// TwinCAT 3 PLC project Base
// ProgramVersion: 3.1.4022.4
// libraries:
//   Tc2_Standard, * (Beckhoff Automation GmbH)
//   Tc2_System, * (Beckhoff Automation GmbH)
//   Tc2_Utilities, * (Beckhoff Automation GmbH)
//   Tc3_IotBase, * (Beckhoff Automation GmbH)
//   Tc3_IotCommunicator, * (Beckhoff Automation GmbH)
//   Tc3_JsonXml, * (Beckhoff Automation GmbH)
//   Tc3_Module, * (Beckhoff Automation GmbH)
// project tree:
//   DUTs/ E_JsonStates.TcDUT, ST_ReceivedData.TcDUT (not stored)
//   GVLs/ CELL_STATE.TcGVL, CELL_WORKING_STATES.TcGVL (not stored), CLAMP_STATE.TcGVL (not stored), CELL_ACTION_STATE.TcGVL (not stored), DATA_SERVICE_STATE.TcGVL, MHS_STATE.TcGVL (not stored), MHS_Registers.TcGVL (not stored)
//   / PlcTask.TcTTO
//   POUs/ FB_Bool_To_Word.TcPOU, FB_Cell_Simu.TcPOU (not stored), FB_InterfaceProfibus.TcPOU, FB_VirtualCell.TcPOU, FB_Word_To_Bool.TcPOU, I_CELL.TcIO (not stored), FB_Cell.TcPOU (not stored), FB_Clamp.TcPOU (not stored), FB_ClampSimulated.TcPOU (not stored), FB_DataService.TcPOU (not stored), FB_InterfaceIO.TcPOU, FB_InterfaceSimulated.TcPOU (not stored), FB_MHS.TcPOU, ITF_Cell.TcIO, JsonSaxHandler.TcPOU, MAIN.TcPOU (not stored), FB_VirtualCellIntWriter.TcPOU
//   POUs/REST API/MHS/ FB_Get.TcPOU, FB_PUT.TcPOU
// real-time tasks:
//   TASK PlcTask: cycle T#10ms, priority 20, ADS port 350
// I/O:
//   DEVICE Device 3 (EtherCAT), AmsNetId 192.168.74.113.4.1
//     Box 1 (CU1128) [CU1128 6x EtherCAT junction]
//       A2_Schaltschrank [EK1100 EtherCAT Coupler (2A E-Bus)]
//         Term 3 (EL2004) [EL2004 4Ch. Dig. Output 24V, 0.5A]
//         Term 4 (EL1004) [EL1004 4Ch. Dig. Input 24V, 3ms]
//         Term 5 (EL2004) [EL2004 4Ch. Dig. Output 24V, 0.5A]
//         Term 6 (EL2004) [EL2004 4Ch. Dig. Output 24V, 0.5A]
//         Term 7 (EL1004) [EL1004 4Ch. Dig. Input 24V, 3ms]
//         Term 8 (EL1004) [EL1004 4Ch. Dig. Input 24V, 3ms]
//         Term 9 (EL2004) [EL2004 4Ch. Dig. Output 24V, 0.5A]
//         Term 10 (EL1004) [EL1004 4Ch. Dig. Input 24V, 3ms]
//         Term 24 (EL9011) [EL9011 End Terminal]
//       A5 [EK1100 EtherCAT Coupler (2A E-Bus)]
//         Term 12 (EL1004) [EL1004 4Ch. Dig. Input 24V, 3ms]
//         Term 13 (EL1004) [EL1004 4Ch. Dig. Input 24V, 3ms]
//         Term 14 (EL2004) [EL2004 4Ch. Dig. Output 24V, 0.5A]
//         Term 15 (EL2004) [EL2004 4Ch. Dig. Output 24V, 0.5A]
//         Term 16 (EL2004) [EL2004 4Ch. Dig. Output 24V, 0.5A]
//         Term 25 (EL9011) [EL9011 End Terminal]
//       Dummy term [CU1128 6x EtherCAT junction - Dev A]
//         Term 18 (EK1100) [EK1100 EtherCAT Coupler (2A E-Bus)]
//           Term 19 (EL1004) [EL1004 4Ch. Dig. Input 24V, 3ms]
//           Term 20 (EL9505) [EL9505 Power supply terminal 5V]
//           Term 21 (EL1124) [EL1124 4Ch. Dig. Input 5V, 10µs, Sensor Power]
//           Term 22 (EL2124) [EL2124 4Ch. Dig. Output 5V, 20mA]
//           Term 26 (EL9011) [EL9011 End Terminal]
//       Term 25 (CU1128-C) [CU1128 6x EtherCAT junction - Dev B]
// variable links:
//   Base/Base Instance <-> Device 3 (EtherCAT)/Box 1 (CU1128)/A2_Schaltschrank/Term 3 (EL2004)
//     PlcTask Outputs/MAIN.fbCellA2.fbClamp.m_bOpen <-> Channel 1/NPSA2
//   Base/Base Instance <-> Device 3 (EtherCAT)/Box 1 (CU1128)/A2_Schaltschrank/Term 4 (EL1004)
//     PlcTask Inputs/MAIN.fbCellA2.fbClamp.m_bIsClosed <-> Channel 1/A2_NPS_Gespannt
//     PlcTask Inputs/MAIN.fbCellA2.fbClamp.m_bIsFull <-> Channel 3/A2_NPS_Ini_Oben
//     PlcTask Inputs/MAIN.fbCellA2.fbClamp.m_bIsOpen <-> Channel 2/A2_NPS_Auf
//   Base/Base Instance <-> Device 3 (EtherCAT)/Box 1 (CU1128)/A2_Schaltschrank/Term 5 (EL2004)
//     PlcTask Outputs/MAIN.fbCellA2.fbInterface.m_bMoveToLoadPos <-> Channel 1/A2_Bestück
//     PlcTask Outputs/MAIN.fbCellA2.fbInterface.m_bMoveToUnloadPos <-> Channel 3/A2_Entnahme
//     PlcTask Outputs/MAIN.fbCellA2.fbInterface.m_bStart <-> Channel 2/A2_Startfreigabe
//     PlcTask Outputs/MAIN.fbCellA2.fbInterface.m_bToStandby <-> Channel 4/A2_Standby
//   Base/Base Instance <-> Device 3 (EtherCAT)/Box 1 (CU1128)/A2_Schaltschrank/Term 7 (EL1004)
//     PlcTask Inputs/MAIN.fbCellA2.fbInterface.m_bFinished <-> Channel 3/A2_Fertig
//     PlcTask Inputs/MAIN.fbCellA2.fbInterface.m_bLoadPos <-> Channel 1/A2_Bestückbereit
//     PlcTask Inputs/MAIN.fbCellA2.fbInterface.m_bRunning <-> Channel 2/A2_Arbeitet
//     PlcTask Inputs/MAIN.fbCellA2.fbInterface.m_bUnloadPos <-> Channel 4/A2_Entnahmebereit
//   Base/Base Instance <-> Device 3 (EtherCAT)/Box 1 (CU1128)/A2_Schaltschrank/Term 8 (EL1004)
//     PlcTask Inputs/MAIN.fbCellA2.fbInterface.m_bEmergencyOff <-> Channel 4/Input
//     PlcTask Inputs/MAIN.fbCellA2.fbInterface.m_bStandby <-> Channel 1/Input
//   Base/Base Instance <-> Device 3 (EtherCAT)/Box 1 (CU1128)/A5/Term 12 (EL1004)
//     PlcTask Inputs/MAIN.fbCellA5.fbInterface.m_bFinished <-> Channel 3/A5_Fertig
//     PlcTask Inputs/MAIN.fbCellA5.fbInterface.m_bLoadPos <-> Channel 1/A5_Bestückbereit
//     PlcTask Inputs/MAIN.fbCellA5.fbInterface.m_bRunning <-> Channel 2/A5_Arbeitet
//     PlcTask Inputs/MAIN.fbCellA5.fbInterface.m_bUnloadPos <-> Channel 4/A5_Entnahmebereit
//   Base/Base Instance <-> Device 3 (EtherCAT)/Box 1 (CU1128)/A5/Term 13 (EL1004)
//     PlcTask Inputs/MAIN.fbCellA5.fbClamp.m_bIsClosed <-> Channel 3/A5_NPS_Zu
//     PlcTask Inputs/MAIN.fbCellA5.fbClamp.m_bIsFull <-> Channel 1/A5_NPS_Ini_Oben
//     PlcTask Inputs/MAIN.fbCellA5.fbClamp.m_bIsOpen <-> Channel 2/A5_NPS_Auf
//   Base/Base Instance <-> Device 3 (EtherCAT)/Box 1 (CU1128)/A5/Term 14 (EL2004)
//     PlcTask Outputs/MAIN.fbCellA5.fbInterface.m_bMoveToLoadPos <-> Channel 1/A5_Bestückposition
//     PlcTask Outputs/MAIN.fbCellA5.fbInterface.m_bMoveToUnloadPos <-> Channel 3/A5_Fahre_Entnahmeposition
//     PlcTask Outputs/MAIN.fbCellA5.fbInterface.m_bStart <-> Channel 2/A5_Startfreigabe
//     PlcTask Outputs/MAIN.fbCellA5.fbInterface.m_bToStandby <-> Channel 4/A5_Fahre_Standby
//   Base/Base Instance <-> Device 3 (EtherCAT)/Box 1 (CU1128)/A5/Term 15 (EL2004)
//     PlcTask Outputs/MAIN.fbCellA5.fbClamp.m_bOpen <-> Channel 1/A5_NPS

CONFIGURATION Base
    RESOURCE PLC ON TwinCAT3
        TASK PlcTask(INTERVAL := T#10ms, PRIORITY := 20);
        PROGRAM MAIN WITH PlcTask : MAIN;
    END_RESOURCE
END_CONFIGURATION

// ---- DUTs/E_JsonStates.TcDUT
{attribute 'qualified_only'}
{attribute 'strict'}
TYPE E_JsonStates :
(
	JSON_STATE_ONSTARTOBJECT1 := 10,
	JSON_STATE_ONKEY_VALUES := 20,
	
	JSON_STATE_ONKEY_ACTIONID := 11,
	JSON_STATE_ONSTRING1 := 12,
	JSON_STATE_ONKEY_WPID := 30,
	JSON_STATE_ONSTRING2 := 40,
	JSON_STATE_ONKEY_WPPLACE := 50,
	JSON_STATE_ONDINT1 := 60,
	JSON_STATE_ONKEY_CELL := 70,
	JSON_STATE_ONUDINT2 := 80,
	JSON_STATE_ONKEY_ACTIONTYPE := 90,
	JSON_STATE_ONUDINT3 := 100,
	JSON_STATE_ONKEY_ACTIONSTATE := 110,
	JSON_STATE_ONUDINT4 := 120,
	JSON_STATE_ONENDOBJECT2 := 1100,
	JSON_STATE_FINISH := 1200
);
END_TYPE

// ---- GVLs/CELL_STATE.TcGVL
{attribute 'qualified_only'}
VAR_GLOBAL
	

			
TYPE 
	CELL_STATE: (e_IDEL, e_WORKING, e_MHS_ACTION, e_ERROR );			
END_TYPE



END_VAR

// ---- GVLs/DATA_SERVICE_STATE.TcGVL
{attribute 'qualified_only'}
VAR_GLOBAL
TYPE
	DATA_SERVICE_STATE: (e_IDLE, e_BUSY, e_FINISHED, e_ERROR);	
END_TYPE
	
END_VAR

// ---- POUs/ITF_Cell.TcIO
INTERFACE ITF_Cell

METHOD GetEmergencyOff : BOOL
VAR_INPUT
END_VAR
END_METHOD

METHOD GetEmergencyStop : BOOL
VAR_INPUT
END_VAR
END_METHOD

METHOD GetFinished : BOOL
VAR_INPUT
END_VAR
END_METHOD

METHOD GetIsRunning : BOOL
VAR_INPUT
END_VAR
END_METHOD

METHOD GetLoadPos : BOOL
VAR_INPUT
END_VAR
END_METHOD

METHOD GetStandby : BOOL
VAR_INPUT
END_VAR
END_METHOD

METHOD GetStartable : BOOL
VAR_INPUT
END_VAR
END_METHOD

METHOD GetUnloadPos : BOOL
VAR_INPUT
END_VAR
END_METHOD

METHOD SetEmergencyOff : BOOL
VAR_INPUT
	b :BOOL;
END_VAR
END_METHOD

METHOD SetEmergencyStop : BOOL
VAR_INPUT
	b :BOOL;
END_VAR
END_METHOD

METHOD SetMoveToLoad : BOOL
VAR_INPUT
	b :BOOL;
END_VAR
END_METHOD

METHOD SetMoveToUnload : BOOL
VAR_INPUT
	b :BOOL;
END_VAR
END_METHOD

METHOD SetStandby : BOOL
VAR_INPUT
	b :BOOL;
END_VAR
END_METHOD

METHOD SetStart : BOOL
VAR_INPUT
	b :BOOL;
END_VAR
END_METHOD

END_INTERFACE

// ---- POUs/FB_Bool_To_Word.TcPOU
FUNCTION_BLOCK FB_Bool_To_Word
VAR_INPUT
//*Hami* Eingang Von FB	als Array Of Bool
	i_Bool : ARRAY [0..15] OF BOOL ;
END_VAR
VAR_OUTPUT
//*Hami* Ausgang Von FB	als UINT
	o_Word : UINT;
END_VAR
VAR
END_VAR

//////////////////////////////////////////////////////////////////////////////////////////////
//*Hami* Diese Funktionsbaustein kann ein Array Of Bool bekommen und in UINT dekodieren
//*Hami* Aufruf von jeder Index von UINT mit UINT.X in Compiler  möglich ist
o_Word.0 := i_Bool[0];
o_Word.1 := i_Bool[1];
o_Word.2 := i_Bool[2];
o_Word.3 := i_Bool[3];
o_Word.4 := i_Bool[4];
o_Word.5 := i_Bool[5];
o_Word.6 := i_Bool[6];
o_Word.7 := i_Bool[7];
o_Word.8 := i_Bool[8];
o_Word.9 := i_Bool[9];
o_Word.10 := i_Bool[10];
o_Word.11 := i_Bool[11];
o_Word.12 := i_Bool[12];
o_Word.13 := i_Bool[13];
o_Word.14 := i_Bool[14];
o_Word.15 := i_Bool[15];
//////////////////////////////////////////////////////////////////////////////////////////////

END_FUNCTION_BLOCK

// ---- POUs/FB_InterfaceProfibus.TcPOU
FUNCTION_BLOCK FB_InterfaceProfibus IMPLEMENTS ITF_Cell
VAR_INPUT

END_VAR
VAR_OUTPUT
END_VAR

VAR
	// Ausgang :engine          AT %IX0.0:        BOOL; 
//Eingänge
//A5Q_Bestuckung AT %QX27.4 : BOOL;
//A5Q_Startfreigabe AT %QX27.5 : BOOL;
//A5Q_Entnahme AT %QX27.6 : BOOL;
//A5Q_Standby AT %QX27.7 : BOOL;
//A5Q_NOT_Aus_Befehl AT %QX28.0 : BOOL;

//INPUTS  A5 Station Variabel : 5V Von Arduino

//A5I_Bestuckbereit_o1 AT %IX43.2 : BOOL;  
//A5I_Arbeitet_o2 AT %IX43.3 : BOOL;
//A5I_Fertig_o3 AT %IX43.4 : BOOL;
//A5I_Storung_o5 AT %IX43.5 : BOOL;
//A5I_NOT_Halt_o6 AT %IX43.6 : BOOL;
//A5I_Pro_Standby_o7 AT %IX43.7 : BOOL;
//A5I_Pro_Standby_o8 AT %IX44.0 : BOOL;
/////////////////////////////////////////////////////////////////////////////////////////////////////////////////
//*Hami* boolesche Eingänge und Ausgänge als innere Variable deklarieren 

//*Hami* innere Eingänge
m_bEmergencyOff  : BOOL; 
m_bEmergencyStop : BOOL;
m_bFinished : BOOL;
m_bRunning : BOOL;
m_bLoadPos  : BOOL; 
m_bUnloadPos  : BOOL; 
m_bStandby : BOOL;
m_bStartable : BOOL;
m_bSoftError  : BOOL;

//*Hami* innere Ausgänge
m_bToEmergencyOff  : BOOL;
m_bToEmergencyStop  : BOOL;
m_bMoveToLoadPos  : BOOL;
m_bMoveToUnloadPos : BOOL;
m_bToStandby  : BOOL;
m_bStart  : BOOL;

//*HAMI* Eingäng und Ausgäng in Form UINT deklarieren zum anpassen Profibus_Dateien
//*HAMI* Die beide müssen zu ProfibusKlemme gelinkt werden

m_wProfibusDataWord AT %I*  : UINT; 
m_wToProfibusDataWord AT %Q*  : UINT;

//*HAMI* Hilf_FBs Deklarieren (Konvertor)

fbBoolToWord : FB_Bool_To_Word;
fbWordToBool : FB_Word_To_Bool;
//*HAMI* Variable für Konvertor FBs ( FB_Bool_to_Word und FB_Word_to_bool )
//*HAMI* i_arrayOfBool Eingänge q_arrayOfBool Ausgänge
i_arrayOfBool : ARRAY [0..15] OF BOOL;
q_arrayOfBool : ARRAY [0..15] OF BOOL;
//*Hami physikalische Eingänge und Ausgänge von Profibus werden drin geschrieben *
i_DataWord : UINT ;
q_DataWord : UINT ;
/////////////////////////////////////////////////////////////////////////////////////////////////////////////////


END_VAR

/////////////////////////////////////////////////////////////////////////////////////////////////////////////////
//*Hami* Aufruf von Hilf_FBs (Konvertor) 
fbBoolToWord();
fbWordToBool();


//hier Wird Mit Hilfe Von Funktion Blocks ( FB_Bool_to_Word und FB_Word_to_bool ) eingänge und Ausgänge angepasst

// Eingänge von Zelle To Bool
i_DataWord := m_wProfibusDataWord ;  //*Hami* Eingang von Profibus in einem hilfsvariabel schreiben
fbWordToBool.i_Word := i_DataWord ; //*Hami* Eingang von Profibus in Eingang von FB_WordToBool schreiben 
i_arrayOfBool :=fbWordToBool.o_Bool ; //*Hami* Ausgang von FB_WordToBool in ein Array of Bool Schreiben 


//*Hami* jeder Index von Array wurde gleich innere Eingänge gestellt 
m_bEmergencyOff := i_arrayOfBool[0];
m_bEmergencyStop := i_arrayOfBool[1]; 
m_bFinished := i_arrayOfBool[2];
m_bRunning := i_arrayOfBool[3];
m_bLoadPos := i_arrayOfBool[4]; 
m_bUnloadPos := i_arrayOfBool[5];   
m_bStandby := i_arrayOfBool[6];
m_bStartable := i_arrayOfBool[7];
m_bSoftError := i_arrayOfBool[8];

//*Hami* Ausgänge von Zelle To Array of Bool 

q_arrayOfBool[0]:= m_bToEmergencyOff ;
q_arrayOfBool[1] := m_bToEmergencyStop;  
q_arrayOfBool[2] := m_bMoveToLoadPos;  
q_arrayOfBool[3] := m_bMoveToUnloadPos; 
q_arrayOfBool[4] := m_bToStandby;  
q_arrayOfBool[5] := m_bStart;

fbBoolToWord.i_Bool := q_arrayOfBool ;//*Hami* Array of Bool in Eingang von fbBoolToWord schreiben
q_DataWord := fbBoolToWord.o_Word ;  //*Hami*  Ausgang von FB_BoolToWord in einem Hilfsvariabel schreiben 
m_wToProfibusDataWord := q_DataWord ; //*Hami* Hilfsvariabel in Ausgang von Profibus Schreiben

/////////////////////////////////////////////////////////////////////////////////////////////////////////////////


// Logik des Interfaces in diesem Fall zurücksetzen der Ausgänge nach erreichen des Ziels 
// Aus Zustandsmaschine Löschen ggf. ??
//IF m_bEmergencyOff THEN
//m_bToEmergencyOff := FALSE;
//END_IF

//IF m_bEmergencyStop THEN
//m_bToEmergencyStop := FALSE;
//END_IF

IF m_bLoadPos THEN
	m_bMoveToLoadPos := FALSE;
END_IF

IF m_bUnloadPos THEN
	m_bMoveToUnloadPos := FALSE;
END_IF

IF m_bStandby THEN
	m_bToStandby := FALSE;
END_IF

IF m_bRunning THEN
	m_bStart := FALSE;
END_IF

METHOD GetEmergencyOff : BOOL
VAR_INPUT
END_VAR
GetEmergencyOff := m_bEmergencyOff;
END_METHOD

METHOD GetEmergencyStop : BOOL
VAR_INPUT
END_VAR
GetEmergencyStop := m_bEmergencyStop;
END_METHOD

METHOD GetFinished : BOOL
VAR_INPUT
END_VAR
GetFinished := m_bFinished;
END_METHOD

METHOD GetIsRunning : BOOL
VAR_INPUT
END_VAR
GetIsRunning := m_bRunning;
END_METHOD

METHOD GetLoadPos : BOOL
VAR_INPUT
END_VAR
GetLoadPos := m_bLoadPos;
END_METHOD

METHOD GetStandby : BOOL
VAR_INPUT
END_VAR
GetStandby := m_bStandby;
END_METHOD

METHOD GetStartable : BOOL
VAR_INPUT
END_VAR
GetStartable := m_bStartable;
END_METHOD

METHOD GetUnloadPos : BOOL
VAR_INPUT
END_VAR
GetUnloadPos := m_bUnloadPos;
END_METHOD

METHOD SetEmergencyOff : BOOL
VAR_INPUT
	b :BOOL;
END_VAR

m_bToEmergencyOff := b;
SetEmergencyOff:=b;
END_METHOD

METHOD SetEmergencyStop : BOOL
VAR_INPUT
	b :BOOL;
END_VAR
m_bToEmergencyStop :=b;

SetEmergencyStop := b;
END_METHOD

METHOD SetMoveToLoad : BOOL
VAR_INPUT
	b :BOOL;
END_VAR
m_bMoveToLoadPos := b;

SetMoveToLoad := b;
END_METHOD

METHOD SetMoveToUnload : BOOL
VAR_INPUT
	b :BOOL;
END_VAR
m_bMoveToUnloadPos := b;

SetMoveToUnload := b;
END_METHOD

METHOD SetStandby : BOOL
VAR_INPUT
	b :BOOL;
END_VAR
m_bToStandby := b;

SetStandby := b;
END_METHOD

METHOD SetStart : BOOL
VAR_INPUT
	b :BOOL;
END_VAR
m_bStart := b;

SetStart := b;
END_METHOD

END_FUNCTION_BLOCK

// ---- POUs/FB_Word_To_Bool.TcPOU
FUNCTION_BLOCK FB_Word_To_Bool
VAR_INPUT
//*Hami* Eingang Von FB	als UINT
	i_Word : UINT;
END_VAR
VAR_OUTPUT
//*Hami* Ausgang Von FB	als Array
	o_Bool : ARRAY [0..15] OF BOOL ;
END_VAR
VAR
END_VAR

//////////////////////////////////////////////////////////////////////////////////////////////
//*Hami* Diese Funktionsbaustein kann ein UINT bekommen und in Array Of Bool dekodieren
//*Hami* Aufruf von jeder Index von UINT mit UINT.X in Compiler  möglich ist
o_Bool[0] := i_Word.0 ;
o_Bool[1] := i_Word.1 ;
o_Bool[2] := i_Word.2 ;
o_Bool[3] := i_Word.3 ;
o_Bool[4] := i_Word.4 ;
o_Bool[5] := i_Word.5 ;	
o_Bool[6] := i_Word.6 ;
o_Bool[7] := i_Word.7 ;
o_Bool[8] := i_Word.8 ;
o_Bool[9] := i_Word.9 ;
o_Bool[10] := i_Word.10 ;
o_Bool[11] := i_Word.11 ;
o_Bool[12] := i_Word.12 ;
o_Bool[13] := i_Word.13 ;
o_Bool[14] := i_Word.14 ;
o_Bool[15] := i_Word.15 ;
//////////////////////////////////////////////////////////////////////////////////////////////

END_FUNCTION_BLOCK

// ---- POUs/FB_VirtualCell.TcPOU
FUNCTION_BLOCK FB_VirtualCell IMPLEMENTS I_CELL
VAR_INPUT
	
END_VAR
VAR_OUTPUT
END_VAR
VAR
	m_csStateRequest : CELL_ACTION_STATE;
	m_csStateRequestOld : CELL_ACTION_STATE;
	m_csState : CELL_ACTION_STATE;
	m_csStateLastCycle : CELL_ACTION_STATE;
	m_csStateLastAction : CELL_ACTION_STATE;
	
	
	m_csSRWorkingState : CELL_WORKING_STATES := CELL_WORKING_STATES.e_FINISHED;
	m_csSRWorkingStateLast : CELL_WORKING_STATES := CELL_WORKING_STATES.e_FINISHED;
	// Eigenschaften
	m_sName : STRING;
	m_bIsDisassemblyCell : BOOL;
	
	m_iWorkpiece : DINT;
	m_sWorkpieceID : STRING;
	

	m_csCellState : CELL_STATE;
	m_csCellStateLast : CELL_STATE;


	
	m_sErrorString : STRING;
	
	// DataServices
	

	m_sConfigString : STRING;
	m_sConfigStringEndGet : STRING  := '_Get.exe';
	m_sConfigStringEndPut : STRING  := '_Put.exe';
	
	// Virtuelle Zellen Verbindung
	fbVirtualCellIntWriter 	: FB_VirtualCellIntWriter;
	fbJson      			: FB_JsonSaxWriter;
	m_sJsonAction 			: STRING;
	m_sActionPath 			: STRING;
	m_sActionName			: STRING;
	m_sActionPathDir 		: STRING   := 'C:\Sysdem\Netzwerklaufwerk_19-0011';
	m_sAMSNetID 			: 	STRING 	:=	'192.168.74.113.1.1';
	
END_VAR

METHOD GetErrorString : STRING
VAR_INPUT
END_VAR
END_METHOD

METHOD GetName : STRING
VAR_INPUT
END_VAR
GetName := m_sName;
END_METHOD

METHOD PUBLIC GetState : INT
VAR_INPUT
	
END_VAR
GetState := CELL_ACTION_STATE.e_Standby;
END_METHOD

METHOD GetWorkpiece : DINT
VAR_INPUT
END_VAR
GetWorkpiece := m_iWorkpiece;
END_METHOD

METHOD IsDisassemblyCell : BOOL
VAR_INPUT
END_VAR
IsDisassemblyCell := FALSE; // Kann keine sein ist virtuell
END_METHOD

METHOD IsError : BOOL
VAR_INPUT
END_VAR
IF m_csCellState = CELL_STATE.e_ERROR THEN
	IsError := TRUE;
END_IF
END_METHOD

METHOD IsIdle : BOOL
VAR_INPUT
END_VAR
IF m_csCellState = CELL_STATE.e_IDEL THEN
	IsIdle := TRUE;
END_IF
END_METHOD

METHOD IsVirtualCell : BOOL
VAR_INPUT
END_VAR
IsVirtualCell :=TRUE;
END_METHOD

METHOD PUBLIC RequestActionState : BOOL
VAR_INPUT
	csStateRequest : CELL_ACTION_STATE;
END_VAR
m_csStateRequest := csStateRequest;
END_METHOD

METHOD RequestWork : BOOL
VAR_INPUT
END_VAR
m_csCellState := CELL_STATE.e_WORKING;
END_METHOD

METHOD SetDisassemblyCell : BOOL
VAR_INPUT
	bIsDisassemblyCell : BOOL;
END_VAR
m_bIsDisassemblyCell := bIsDisassemblyCell;
END_METHOD

METHOD SetGetDataServiceEnable : BOOL
VAR_INPUT
END_VAR

SetGetDataServiceEnable := FALSE;
END_METHOD

METHOD SetName : BOOL
VAR_INPUT
	sName :string ;
END_VAR
m_sName := sName;
END_METHOD

METHOD SetPutDataServiceEnable : BOOL
VAR_INPUT
END_VAR

SetPutDataServiceEnable := FALSE;
END_METHOD

METHOD SetVirtualCell : BOOL
VAR_INPUT
END_VAR
END_METHOD

METHOD SetWorkpiece : BOOL
VAR_INPUT
	iWorkpiece : DINT;
	sWorkpieceID : STRING;
END_VAR
m_iWorkpiece := iWorkpiece;
m_sWorkpieceID := sWorkpieceID;
END_METHOD

METHOD PUBLIC StateMachine : BOOL
VAR_INPUT
END_VAR

//Zellen Zustandsmaschine

CASE m_csCellState OF 
	CELL_STATE.e_IDEL:
			
	
		;
 	CELL_STATE.e_MHS_ACTION;
		//SubRoutine für Aktion beim beladen aktuell leer da keine MHS für eine virtuelle Zelle verfügbar sind 
		;
	CELL_STATE.e_WORKING:
		//SubRoutine zum Durchführen einer Bearbeitung
			//Erstellen des Json-Strings für die Datei		
			fbJson.ResetDocument();
		
			fbJson.StartObject();
            fbJson.AddKey('Name');
			fbJson.AddString(m_sName);
			fbJson.AddKey('WPID');
			fbJson.AddString(m_sWorkpieceID);			
			fbJson.EndObject();
			m_sJsonAction := fbJson.GetDocument();
		
			// Phad der Schnittstellen-Datei
			m_sActionPath := CONCAT (m_sActionPathDir,'\');
			m_sActionPath := CONCAT (m_sActionPath, m_sName);
			m_sActionPath := CONCAT (m_sActionPath, '_');
			m_sActionPath := CONCAT (m_sActionPath, m_sWorkpieceID);
			m_sActionPath := CONCAT (m_sActionPath, '.json');
			
			// Name der Schnittstellen-Datei
			m_sActionName := CONCAT (m_sName, '_');
			m_sActionName := CONCAT (m_sActionName, m_sWorkpieceID);
			m_sActionName := CONCAT (m_sActionName, '.json');
			
			// Nächster Schritt SubRoutine Starten um das Schreiben auszugühren
			IF NOT (CELL_STATE.e_WORKING = m_csCellStateLast) THEN  
				m_csSRWorkingState := CELL_WORKING_STATES.e_START;
			END_IF

			
	CASE m_csSRWorkingState OF
			
			CELL_WORKING_STATES.e_START:
				fbVirtualCellIntWriter.buffRead := m_sJsonAction; // Inhalt der Datei übergeben
				fbVirtualCellIntWriter.sDestPathName := m_sActionPath; // Pfad der Datei
				fbVirtualCellIntWriter.sDestNetId := m_sAMSNetID;// Net Id des HostPC
				fbVirtualCellIntWriter.tTimeOut := DEFAULT_ADS_TIMEOUT;// Fehlerzeit
				fbVirtualCellIntWriter.bExecute := TRUE;// Positive flanke zum Starten
				IF fbVirtualCellIntWriter.bError THEN//
					m_csCellState := CELL_STATE.e_ERROR;
				END_IF
				IF fbVirtualCellIntWriter.bBusy THEN // Der Funktionsblock aufgehört hat zu arbeiten nächster Schritt ggf. das vorhanden sein der Datei prüfen 
					
					m_csSRWorkingState := CELL_WORKING_STATES.e_WORKING;
				END_IF
				

				
			CELL_WORKING_STATES.e_WORKING:	
				fbVirtualCellIntWriter.bExecute := FALSE; // Nur positive Flanke
				IF NOT(fbVirtualCellIntWriter.bBusy) THEN // Der Funktionsblock aufgehört hat zu arbeiten nächster Schritt ggf. das vorhanden sein der Datei prüfen 
					
					m_csSRWorkingState := CELL_WORKING_STATES.e_FINISHED;
				END_IF
				
			CELL_WORKING_STATES.e_FINISHED:
				m_iWorkpiece := 0;
				m_sWorkpieceID := 'Empty';
				m_csCellState := CELL_STATE.e_IDEL;
			
		END_CASE
		
	CELL_STATE.e_ERROR:
			;
END_CASE

m_csCellStateLast := m_csCellState;
fbVirtualCellIntWriter();
fbVirtualCellIntWriter.StateMachine();
END_METHOD

METHOD StateMachineProfibus : BOOL
VAR_INPUT
END_VAR
END_METHOD

END_FUNCTION_BLOCK

// ---- POUs/FB_VirtualCellIntWriter.TcPOU
FUNCTION_BLOCK FB_VirtualCellIntWriter
VAR_INPUT
     
        sDestNetId              : T_AmsNetId;(* TwinCAT network address of the destination file *)
        sDestPathName           : T_MaxString; (* Destination file path and name *)
        bExecute                : BOOL; (* Rising edge start fb execution *)
        tTimeOut                : TIME := DEFAULT_ADS_TIMEOUT;(* Max. ADS timeout time *)
		buffRead                : STRING;// ARRAY[1..1000] OF BYTE;(* Buffer *)
END_VAR
VAR_OUTPUT
        bBusy                   :BOOL;(* TRUE => File copy execution in progress, FALSE => File copy execution idle *)
 		bError                  :BOOL;(* TRUE => Error, FALSE => No error *)
 		nErrId                  :UDINT;(* Error code *)
END_VAR
VAR
        fbFileOpen              :FB_FileOpen;
        fbFileClose             :FB_FileClose;
        fbFileRead              :FB_FileRead;
        fbFileWrite             :FB_FileWrite;

        hSrcFile                :UINT   := 0;(* File handle of the source file *)
 		hDestFile               :UINT   := 0;(* File handle of the destination file *)

        Step                    :DWORD;
        RisingEdge              :R_TRIG;

        
 		cbReadLength            :UDINT := 0;
END_VAR

METHOD StateMachine : BOOL
VAR_INPUT
END_VAR
RisingEdge(CLK:=bExecute);

CASE Step OF
        0:      (* Idle state *)
         IF RisingEdge.Q THEN
                        bBusy := TRUE;
                        bError:= FALSE;
                        nErrId:=0;
                        Step := 1;
                        cbReadLength:=0;
                        hSrcFile:=0;
                        hDestFile:=0;
                END_IF



        1:      (* Open destination file *)
         fbFileOpen( bExecute := FALSE );
                fbFileOpen( sNetId := sDestNetId, sPathName := sDestPathName,
                        nMode := FOPEN_MODEWRITE OR FOPEN_MODEBINARY,
                        ePath := PATH_GENERIC, tTimeout := tTimeOut, bExecute := TRUE );
                Step := Step+1;
        2:
                fbFileOpen( bExecute := FALSE );
                IF NOT fbFileOpen.bBusy THEN
                        IF fbFileOpen.bError THEN
                                nErrId := fbFileOpen.nErrId;
                                bError := TRUE;
                                Step := 50;
                        ELSE
                                hDestFile := fbFileOpen.hFile;
                                Step := Step + 1;
                        END_IF
                END_IF

        3:      (* Write data to destination file *)
         fbFileWrite( bExecute := FALSE );
                fbFileWrite( sNetId:=sDestNetId, hFile:=hDestFile,
                        pWriteBuff:= ADR(buffRead), cbWriteLen:= INT_TO_UDINT(LEN(buffRead)),
                        bExecute:=TRUE, tTimeout:=tTimeOut );
                Step := Step + 1;
				
        4:
                fbFileWrite( bExecute := FALSE );
                IF NOT fbFileWrite.bBusy THEN
                        IF fbFileWrite.bError THEN
                                nErrId := fbFileWrite.nErrId;
                                bError := TRUE;
                                Step := 50;
                        ELSE
                                 Step := 50;(* Cleanup: close the destination and source files *)
                         
                        
                        END_IF
                END_IF

        30:     (* Close the destination file *)
         fbFileClose( bExecute := FALSE );
                fbFileClose( sNetId:=sDestNetId, hFile:=hDestFile, bExecute:=TRUE, tTimeout:=tTimeOut );
                Step := Step + 1;
        31:
                fbFileClose( bExecute := FALSE );
                IF NOT fbFileClose.bBusy THEN
                        IF fbFileClose.bError THEN
                                nErrId := fbFileClose.nErrId;
                                bError := TRUE;
                        END_IF
                        Step := 50;
                        hDestFile := 0;
                END_IF

        40: (* Close source file *)
         fbFileClose( bExecute := FALSE );
               // fbFileClose( sNetId:=sSrcNetId, hFile:=hSrcFile, bExecute:=TRUE, tTimeout:=tTimeOut );
                Step := Step + 1;
        41:
                fbFileClose( bExecute := FALSE );
                IF NOT fbFileClose.bBusy THEN
                        IF fbFileClose.bError THEN
                                nErrId := fbFileClose.nErrId;
                                bError := TRUE;
                        END_IF
                        Step := 50;
                        hSrcFile := 0;
                END_IF

        50: (* Error or ready => Cleanup *)
         IF ( hDestFile <> 0 ) THEN
                        Step := 30; (* Close the destination file*)
         ELSIF (hSrcFile <> 0 ) THEN
                        Step := 40; (* Close the source file *)
         ELSE
                        Step := 0;      (* Ready *)
                        bBusy := FALSE;
                END_IF

END_CASE
END_METHOD

END_FUNCTION_BLOCK

// ---- POUs/FB_InterfaceIO.TcPOU
FUNCTION_BLOCK FB_InterfaceIO IMPLEMENTS ITF_Cell
VAR_INPUT

END_VAR
VAR_OUTPUT
END_VAR


	// Ausgang :engine          AT %IX0.0:        BOOL; 
//Eingänge
//A5Q_Bestuckung AT %QX27.4 : BOOL;
//A5Q_Startfreigabe AT %QX27.5 : BOOL;
//A5Q_Entnahme AT %QX27.6 : BOOL;
//A5Q_Standby AT %QX27.7 : BOOL;
//A5Q_NOT_Aus_Befehl AT %QX28.0 : BOOL;

//INPUTS  A5 Station Variabel : 5V Von Arduino

//A5I_Bestuckbereit_o1 AT %IX43.2 : BOOL;  
//A5I_Arbeitet_o2 AT %IX43.3 : BOOL;
//A5I_Fertig_o3 AT %IX43.4 : BOOL;
//A5I_Storung_o5 AT %IX43.5 : BOOL;
//A5I_NOT_Halt_o6 AT %IX43.6 : BOOL;
//A5I_Pro_Standby_o7 AT %IX43.7 : BOOL;
//A5I_Pro_Standby_o8 AT %IX44.0 : BOOL;
VAR
m_bEmergencyOff AT %I* : BOOL;
m_bEmergencyStop AT %I* : BOOL;
m_bFinished AT %I* : BOOL;
m_bRunning AT %I* : BOOL;
m_bLoadPos  AT %I* : BOOL; 
m_bUnloadPos  AT %I* : BOOL; 
m_bStandby AT %I* : BOOL;
m_bStartable AT %I* : BOOL;
m_bSoftError AT %I* : BOOL;
// Ausgang :engine          AT %QX0.0:        BOOL; 
// Ausgänge
m_bToEmergencyOff AT %Q* : BOOL;
m_bToEmergencyStop AT %Q* : BOOL;
m_bMoveToLoadPos AT %Q* : BOOL;
m_bMoveToUnloadPos AT %Q* : BOOL;
m_bToStandby AT %Q* : BOOL;
m_bStart AT %Q* : BOOL;

END_VAR

// Logik des Interfaces in diesem Fall zurücksetzen der Ausgänge nach erreichen des Ziels 
// Aus Zustandsmaschine Löschen ggf. ??
//IF m_bEmergencyOff THEN
//m_bToEmergencyOff := FALSE;
//END_IF

//IF m_bEmergencyStop THEN
//m_bToEmergencyStop := FALSE;
//END_IF

IF m_bLoadPos THEN
	m_bMoveToLoadPos := FALSE;
END_IF

IF m_bUnloadPos THEN
	m_bMoveToUnloadPos := FALSE;
END_IF

IF m_bStandby THEN
	m_bToStandby := FALSE;
END_IF

IF m_bRunning THEN
	m_bStart := FALSE;
END_IF

METHOD GetEmergencyOff : BOOL
VAR_INPUT
END_VAR
GetEmergencyOff := m_bEmergencyOff;
END_METHOD

METHOD GetEmergencyStop : BOOL
VAR_INPUT
END_VAR
GetEmergencyStop := m_bEmergencyStop;
END_METHOD

METHOD GetFinished : BOOL
VAR_INPUT
END_VAR
GetFinished := m_bFinished;
END_METHOD

METHOD GetIsRunning : BOOL
VAR_INPUT
END_VAR
GetIsRunning := m_bRunning;
END_METHOD

METHOD GetLoadPos : BOOL
VAR_INPUT
END_VAR
GetLoadPos := m_bLoadPos;
END_METHOD

METHOD GetStandby : BOOL
VAR_INPUT
END_VAR
GetStandby := m_bStandby;
END_METHOD

METHOD GetStartable : BOOL
VAR_INPUT
END_VAR
GetStartable := m_bStartable;
END_METHOD

METHOD GetUnloadPos : BOOL
VAR_INPUT
END_VAR
GetUnloadPos := m_bUnloadPos;
END_METHOD

METHOD SetEmergencyOff : BOOL
VAR_INPUT
	b :BOOL;
END_VAR

m_bToEmergencyOff := b;
SetEmergencyOff:=b;
END_METHOD

METHOD SetEmergencyStop : BOOL
VAR_INPUT
	b :BOOL;
END_VAR
m_bToEmergencyStop :=b;

SetEmergencyStop := b;
END_METHOD

METHOD SetMoveToLoad : BOOL
VAR_INPUT
	b :BOOL;
END_VAR
m_bMoveToLoadPos := b;

SetMoveToLoad := b;
END_METHOD

METHOD SetMoveToUnload : BOOL
VAR_INPUT
	b :BOOL;
END_VAR
m_bMoveToUnloadPos := b;

SetMoveToUnload := b;
END_METHOD

METHOD SetStandby : BOOL
VAR_INPUT
	b :BOOL;
END_VAR
m_bToStandby := b;

SetStandby := b;
END_METHOD

METHOD SetStart : BOOL
VAR_INPUT
	b :BOOL;
END_VAR
m_bStart := b;

SetStart := b;
END_METHOD

END_FUNCTION_BLOCK

// ---- POUs/FB_MHS.TcPOU
FUNCTION_BLOCK FB_MHS


VAR
	m_csStateRequest : MHS_STATE;
	m_csStateRequestOld : MHS_STATE;
	m_csState : MHS_STATE;
	m_csStateLastCycle : MHS_STATE;
	m_csStateLastAction : MHS_STATE;
	m_Name : STRING;	
	// Von SystemDemonstratorApp kommend
	m_iWorkpiece : DINT; 
	m_iCell : DINT;
	m_iRequest: DINT;
	// Von SystemDemonstratorApp kommend angenommen
	m_iWorkpieceAccepted : DINT; 
	m_iCellAccepted : DINT;
	m_iRequestAccepted: DINT;
	
	// Von PLC kommend 
	m_iMachineFree : DINT;	
	
	
	//Von MiR kommend
	m_iRequestMachineFree : DINT;
	m_iActionTerminated : DINT;	
	
	
	
	// Zustand der Zelle die Beladen oder Entladen werden soll
	m_eCurrentCellState : CELL_ACTION_STATE;
	m_eNeededCellState : CELL_ACTION_STATE;
	m_bNeededCellStatePending : BOOL;
	
	aMHS : ARRAY [1..20] OF DINT; // Interface API-Array
	
	
	m_iSimulationsTimer : DINT;


			////////////////////////////////////////////*Hami*////////////////////////////////////////////////////////////

//*Hami* RisingEdge zum Ausführung von REST_API FBs	
	bGet, bPut   			: BOOL;
	

//*Hami* FB Client initialisieren (Das wir in FB_GET und FB_PUT augerufen) 
//*Hami* http://mir.com/api/v2.0.0/registers/x für die Ardresse x=[1 bis 200] gibts ein Register , die mit JSON_String geschrieben werden können
//*Hami* JSON_Strings für jedes Register sieht so aus :	{"value": x,"label": "string"}

	fbClient				:  FB_IotHttpClient :=(sHostName:='mir.com',
								  	bKeepAlive:=TRUE, tConnectionTimeout:=T#5S);
									
//*Hami* Array von REST_API FBs (PUT zum Schreiben , GET zum Lesen)								
	fbGet					:ARRAY [11..20] OF FB_Get; 
	fbPut					:ARRAY [1..10] OF FB_PUT; 

			////////////////////////////////////////////*Hami*////////////////////////////////////////////////////////////
END_VAR

StateMachine();

			/////////////////////////////////////////////////*Hami*//////////////////////////////////////////////////////////////////
///////////////////////////////*Hami*  lesen und schreiben Dateien an REST API///////////////////////////////////////////
//*Hami* HostPort einstellen , wenn es nötig ist
	
	//IF NOT fbClient.bConfigured THEN 
	//fbClient.nHostPort:= 80;
	//END_IF 

//*Hami* Interface API-Array(aMHS[1..10] zum schreiben in Registers von MHS , aMHS[11..20] zum lesen von Registers )

fbPut[1].value := aMHS[1];
fbPut[2].value := aMHS[2];
fbPut[3].value := aMHS[3];
fbPut[4].value := aMHS[4];
fbPut[5].value := aMHS[5];

//*Hami* init client parameters at startup (für jedes Register gibt es ein Funktion_Block)		
////////////////////////////////////////1/////////////////////////////////////////////////		

IF fbClient.bConfigured THEN 
		fbGet[11](bSend:=bGet,sURi := '/api/v2.0.0/registers/11', fbClient:=fbClient);
		fbPut[1](bSend:=bPut,sURi := '/api/v2.0.0/registers/1',DefaultMessage := '{"value": x}', fbClient:=fbClient);
END_IF
fbClient.Execute();
///////////////////////////////////////2//////////////////////////////////////////////////		

IF fbClient.bConfigured THEN 
		fbGet[12](bSend:=bGet,sURi := '/api/v2.0.0/registers/12', fbClient:=fbClient);
		fbPut[2](bSend:=bPut,sURi := '/api/v2.0.0/registers/2',DefaultMessage := '{"value": x}', fbClient:=fbClient);
END_IF
fbClient.Execute();
///////////////////////////////////////3//////////////////////////////////////////////////		

IF fbClient.bConfigured THEN 
		fbGet[13](bSend:=bGet,sURi := '/api/v2.0.0/registers/13', fbClient:=fbClient);
		fbPut[3](bSend:=bPut,sURi := '/api/v2.0.0/registers/3',DefaultMessage := '{"value": x}', fbClient:=fbClient);
END_IF
fbClient.Execute();
///////////////////////////////////////4//////////////////////////////////////////////////		

IF fbClient.bConfigured THEN 
		fbGet[14](bSend:=bGet,sURi := '/api/v2.0.0/registers/14', fbClient:=fbClient);
		fbPut[4](bSend:=bPut,sURi := '/api/v2.0.0/registers/4',DefaultMessage := '{"value": x}', fbClient:=fbClient);
END_IF
fbClient.Execute();
///////////////////////////////////////5//////////////////////////////////////////////////		

IF fbClient.bConfigured THEN 
		fbGet[15](bSend:=bGet,sURi := '/api/v2.0.0/registers/15', fbClient:=fbClient);
		fbPut[5](bSend:=bPut,sURi := '/api/v2.0.0/registers/5',DefaultMessage := '{"value": x , "label":"kann hier geschrieben werden"}', fbClient:=fbClient);
END_IF
fbClient.Execute();

//*Hami* SET Registers Connection with MHS


aMHS[11] := fbGet[11].value;
aMHS[12] := fbGet[12].value;
aMHS[13] := fbGet[13].value;
aMHS[14] := fbGet[14].value;
aMHS[15] := fbGet[15].value;

			/////////////////////////////////////////////////*Hami*//////////////////////////////////////////////////////////////////

METHOD GetActionFinished : BOOL
VAR_INPUT
END_VAR
IF m_csState = MHS_STATE.e_AKTION_FINISHED THEN
	GetActionFinished := TRUE;
ELSE
	GetActionFinished := FALSE;
END_IF
END_METHOD

METHOD GetCurrentCellForAction : DINT
VAR_INPUT
END_VAR
GetCurrentCellForAction := m_iCellAccepted;
END_METHOD

METHOD GetState : BOOL
VAR_INPUT
END_VAR
END_METHOD

METHOD NeededCellStatePending : BOOL
VAR_INPUT
END_VAR
NeededCellStatePending := m_bNeededCellStatePending;
m_bNeededCellStatePending := FALSE;
END_METHOD

METHOD RequestAction : BOOL
VAR_INPUT
	
	iWorkpiece : DINT; 
	iCell : DINT;
	bRequest : DINT;
END_VAR

m_iWorkpiece :=  iWorkpiece;
m_iCell := iCell;
m_iRequest := bRequest;
END_METHOD

METHOD RequestState : BOOL
VAR_INPUT
END_VAR
END_METHOD

METHOD SendNeededToCell : CELL_ACTION_STATE
VAR_INPUT
END_VAR
SendNeededToCell := m_eNeededCellState;
END_METHOD

METHOD SetClampIsOpen : BOOL
VAR_INPUT
iClampIsOpen : DINT;	

END_VAR
//IF iClampIsOpen > 0 THEN
//	m_iClampIsOpen := 1;
//	m_iClampIsClose := 0;
//ELSE
//	m_iClampIsOpen := 0;
//	m_iClampIsClose := 1;	
//END_IF
END_METHOD

METHOD SetDoorIsOpen : BOOL
VAR_INPUT
	iDoorIsOpen :DINT;
END_VAR
//IF iDoorIsOpen > 0 THEN
//	m_iDoorIsOpen := 1;
//	m_iDoorIsClose := 0;
//ELSE
//	m_iDoorIsOpen := 0;
//	m_iDoorIsClose := 1;	
//END_IF
END_METHOD

METHOD SetMachineFree : BOOL
VAR_INPUT
	iMachineFree:DINT;
END_VAR
m_iMachineFree := iMachineFree;
END_METHOD

METHOD SetStateCurrentMachineForAction : BOOL
VAR_INPUT
	eCurrentCellState :CELL_ACTION_STATE;
END_VAR
m_eCurrentCellState := eCurrentCellState;

SetStateCurrentMachineForAction := TRUE;
END_METHOD


METHOD StateMachine : BOOL
VAR_INPUT
END_VAR

VAR

END_VAR

	// VOM MHS

	//{define Simulated}
	{define MHSConnected}
	
	{IF defined (MHSConnected)}
 	m_iRequestMachineFree   := aMHS[11];
	m_iActionTerminated :=  aMHS[12];
	{END_IF}
	// PLC interne Variablen
	//m_iDoorIsOpen : DINT;	
	//m_iClampIsOpen : DINT;
	//m_iClampIsClose : DINT;	
	//m_iDoorIsClose : DINT;


	
	
CASE m_csState OF

MHS_STATE.e_IDLE: 

	IF m_iWorkpiece > 0 AND m_iCell > 0 AND m_iRequest > 0 THEN
		m_iWorkpieceAccepted := m_iWorkpiece;  
		m_iCellAccepted := m_iCell;
		m_iRequestAccepted:= m_iRequest; 	
	END_IF

	IF m_iWorkpieceAccepted > 0 AND m_iCellAccepted > 0 AND m_iRequestAccepted = 2 THEN
		aMHS[1] := m_iWorkpieceAccepted;
		aMHS[2] := m_iCellAccepted;
		aMHS[3] := m_iRequestAccepted;
		m_iWorkpiece := 0;
 		m_iCell := 0;
		m_iRequest := 0;
		m_csState := MHS_STATE.e_PGO_POS;	
	END_IF
	IF m_iWorkpieceAccepted > 0 AND m_iCellAccepted > 0 AND m_iRequestAccepted = 1 THEN
		aMHS[1] := m_iWorkpieceAccepted;
		aMHS[2] := m_iCellAccepted;
		aMHS[3] := m_iRequestAccepted;
		m_iWorkpiece := 0;
 		m_iCell := 0;
		m_iRequest := 0;
		m_csState := MHS_STATE.e_GGO_POS;	
	END_IF
	// Löschen dieser Anforderung
	m_iRequestAccepted := 0;


// SUBROUTINE WP in Maschine bringen	  
MHS_STATE.e_PGO_POS:
	
 	IF m_iRequestMachineFree > 0 THEN
		m_eNeededCellState := CELL_ACTION_STATE.e_LoadPos;
		m_bNeededCellStatePending := TRUE;
		m_csState := MHS_STATE.e_PWAIT_DOOR;
	END_IF
	

MHS_STATE.e_PWAIT_DOOR:	
  	IF  m_eCurrentCellState = CELL_ACTION_STATE.e_LoadPos THEN
		//aMHS[3] := 0;//m_iRequest;
		m_iMachineFree := 1;
		m_csState := MHS_STATE.e_PWAIT_CLAMP;
	END_IF

MHS_STATE.e_PWAIT_CLAMP:
		m_csState := MHS_STATE.e_PPUT_WP;
	

MHS_STATE.e_PPUT_WP:
		m_csState := MHS_STATE.e_PCLOSE_CLAMP;
		
 MHS_STATE.e_PCLOSE_CLAMP:
			m_csState := MHS_STATE.e_PLEAFE_MACHINE;
	 
MHS_STATE.e_PLEAFE_MACHINE:
 	IF m_iActionTerminated > 0 THEN
		m_csState := MHS_STATE.e_AKTION_FINISHED;
	END_IF	

// SUBROUTINE WP aus Maschine holen	  
MHS_STATE.e_GGO_POS:
 	IF m_iRequestMachineFree > 0 THEN
		m_eNeededCellState := CELL_ACTION_STATE.e_UnLoadPos;
		m_bNeededCellStatePending := TRUE;
		m_csState := MHS_STATE.e_GWAIT_DOOR;
	END_IF

	
MHS_STATE.e_GWAIT_DOOR:
  	IF  m_eCurrentCellState = CELL_ACTION_STATE.e_UnLoadPos THEN
		m_iMachineFree := 1;
		//aMHS[3] := 0;//m_iRequest;
		m_csState := MHS_STATE.e_GWAIT_CLAMP;
	END_IF

MHS_STATE.e_GWAIT_CLAMP:
	//IF m_iClampIsOpen > 0 THEN
		m_csState := MHS_STATE.e_GGET_WP;
	//END_IF
MHS_STATE.e_GGET_WP:
	//IF 	m_iClampCloseRequest > 0 THEN
		m_csState := MHS_STATE.e_GCLOSE_CLAMP;
	//END_IF
 MHS_STATE.e_GCLOSE_CLAMP:
 	//IF m_iClampIsClose > 0 THEN
			m_csState := MHS_STATE.e_GLEAFE_MACHINE;	 
 	//END_IF
MHS_STATE.e_GLEAFE_MACHINE:
	
 	IF m_iActionTerminated > 0 THEN
		aMHS[3] := 0;//m_iRequest;
		m_csState := MHS_STATE.e_AKTION_FINISHED;
	END_IF		

MHS_STATE.e_AKTION_FINISHED:
	m_csState := MHS_STATE.e_IDLE;
	m_iMachineFree := 0;
	
MHS_STATE.e_ERROR:
	
ELSE
	m_csState := MHS_STATE.e_ERROR;
 
END_CASE
{IF defined (MHSConnected)}
aMHS[4] :=  m_iMachineFree; 
{END_IF}
END_METHOD

END_FUNCTION_BLOCK

// ---- POUs/REST API/MHS/FB_Get.TcPOU
//*Hami*
//*Hami* Das Funktion Block liest ein JSON_String von der Ardesse sURi und Schreibt es in OUTPUT value
FUNCTION_BLOCK FB_Get
VAR_INPUT
	bSend				: BOOL;
	sURi : STRING;
	
END_VAR
VAR_IN_OUT
	fbClient			: FB_IotHttpClient;
END_VAR
VAR_OUTPUT
	bBusy				: BOOL;
	bError				: BOOL;
	id					: DINT;
	r_value 			: LREAL;
	value				: DINT;
END_VAR
VAR
	fbHeader: FB_IotHttpHeaderFieldMap ;
	fbRequest			: FB_IotHttpRequest;
	fbJson				: FB_JsonDomParser;
	nState				: UDINT;
	RisingEdge			: R_TRIG;
	
	bGetContentResult	: BOOL;
	sContent			: STRING(511);
	
	bGetJsonResult		: BOOL;
	jsonDoc				: SJsonValue;
	jsonVal				: SJsonValue;
	jsonID				: SJsonValue;
	
	sResultValue		: STRING;
	
	nReqCount			: UDINT;	
	nResCount			: UDINT;
	nValidResCount		: UDINT;
	nErrCount			: UDINT;
	b : BOOL ;
	stReceivedData : ST_ReceivedData ;
	bOnce: BOOL := TRUE ;
	
END_VAR

//*Hami* Authorization einstellen	
	fbHeader.AddField('Authorization', 'Basic RmVsaXg6OGM2OTc2ZTViNTQxMDQxNWJkZTkwOGJkNGRlZTE1ZGZiMTY3YTljODczZmM0YmI4YTgxZjZmMmFiNDQ4YTkxOA==', FALSE);
	fbHeader.AddField('Accept-Language', 'de_DE' , FALSE);
	


//*Hami* hier werden Dateien von sURi als JSON gelesen 
	//RisingEdge(CLK:= bSend );
CASE nState OF
0:	
	//IF RisingEdge.Q THEN 
		IF fbRequest.SendRequest(sURi:=sURi, fbClient:=fbClient, eRequestType:=ETcIotHttpRequestType.HTTP_GET,0, 0, fbHeader) THEN	
	//IF fbRequest.GetJsonDomContent(sURi := sURi , fbClient := fbClient , eRequestType:=ETcIotHttpRequestType.HTTP_GET ,fbJson := fbJson,0) THEN				
			nState:= 1;
			nReqCount:= nReqCount+1;
			bBusy:= TRUE;
			bError:= FALSE;
		END_IF					
	//END_IF
	
//*Hami* hier wird Json_String dekodiert .id und value sind lesbar wenn dateien richtig dekodiert werden
1:
	IF NOT fbRequest.bBusy THEN
		bError:= TRUE;
		IF NOT fbRequest.bError THEN
				bGetContentResult:= fbRequest.GetContent(pContent:= ADR(sContent), nContentSize:= SIZEOF(sContent), bSetNullTermination:= TRUE);
			IF fbRequest.nStatusCode >= 200 AND fbRequest.nStatusCode < 300 THEN
				bGetJsonResult:= FALSE;
				jsonDoc:= fbRequest.GetJsonDomContent(fbJson);
				IF jsonDoc <> 0 THEN
					bGetJsonResult:= TRUE;
					IF fbJson.HasMember(jsonDoc, 'id')  THEN
						jsonID:= fbJson.FindMember(jsonDoc, 'id');
						id := fbJson.GetInt(jsonID);
						IF fbJson.HasMember(jsonDoc, 'value')  THEN
							jsonVal := fbJson.FindMember(jsonDoc, 'value');
							r_value := fbJson.GetDouble(jsonVal);
							value := LREAL_TO_DINT(r_value);
							nValidResCount:= nValidResCount+1;
							bError:= FALSE;						
							IF fbJson.IsString(jsonVal) THEN							
								sResultValue:= fbJson.GetString(jsonVal);									
							END_IF
						END_IF		
					END_IF
				END_IF							
				nResCount:= nResCount+1;			
			END_IF
		END_IF
		nState:= 0;
		bBusy:= FALSE;
		IF bError THEN
			nErrCount:= nErrCount+1;
		END_IF
	END_IF  	
END_CASE

END_FUNCTION_BLOCK

// ---- POUs/REST API/MHS/FB_PUT.TcPOU
//*Hami* 
//*Hami* Das Funktion Block Schreibt INPUT value in Adresse sURi als JSON_String
FUNCTION_BLOCK FB_PUT
VAR_INPUT
	bSend				: BOOL;
	value		 		: DINT ;
	sURi 		 		: STRING;
	DefaultMessage 		: STRING(255);
END_VAR
VAR_IN_OUT
	fbClient			: FB_IotHttpClient;
END_VAR
VAR_OUTPUT
	bBusy				: BOOL;
	bError				: BOOL;
END_VAR
VAR
	fbRequest			: FB_IotHttpRequest;
	fbHeader			: FB_IotHttpHeaderFieldMap;
	fbJson				: FB_JsonDomParser;
	nState				: UDINT;
	RisingEdge			: R_TRIG;

	bGetContentResult	: BOOL;
	sContent			: STRING(511);
	
	bGetJsonResult		: BOOL;
	jsonDoc				: SJsonValue;
	jsonTitle			: SJsonValue;
	jsonVal				: SJsonValue;
	bResultValue		: BOOL;
	
	nReqCount			: UDINT;	
	nResCount			: UDINT;
	nValidResCount		: UDINT;
	nErrCount			: UDINT;
	bOnce				: BOOL:= TRUE;
	sMessage			: STRING(255);
	JsonStringValue		: SJsonValue;
	s_iRegister 		: STRING ;
	ss_iRegister		: STRING ;
END_VAR

//*Hami* value in Jsonvalue (Das ist Externe Datentype im ersten Ordner) schreiben (sMassage ist ein Json_String )
s_iRegister := DINT_TO_STRING(value);
sMessage := REPLACE(DefaultMessage,s_iRegister,1,11);
JsonStringValue := fbJson.ParseDocument(sMessage);

/////////////////////////////////////////////////////////////////////////////
	// RisingEdge(CLK:= bSend);

//*Hami* Authorization einstellen	
	
	//IF RisingEdge.Q  THEN
	fbHeader.AddField('Authorization', 'Basic RmVsaXg6OGM2OTc2ZTViNTQxMDQxNWJkZTkwOGJkNGRlZTE1ZGZiMTY3YTljODczZmM0YmI4YTgxZjZmMmFiNDQ4YTkxOA==', FALSE);
	fbHeader.AddField('Accept-Language', 'de_DE' , FALSE);
	// END_IF
CASE nState OF
0:	
	//IF RisingEdge.Q THEN 
	
	//*Hami* hier werden die Dateien als JSON in sRUi geschrieben 
		IF fbRequest.SendJsonDomRequest(sUri:= sURi , fbClient:=fbClient, eRequestType:=ETcIotHttpRequestType.HTTP_PUT, fbJson := fbJson, fbHeader:=fbHeader) THEN				
			nState:= 1;
			nReqCount:= nReqCount+1;
			bBusy:= TRUE;
			bError:= FALSE;
		END_IF					
	//END_IF
	
	//*Hami* hier werden wieder geschriebene Dataeien von sURi gelesen
1:
	IF NOT fbRequest.bBusy THEN
		bError:= TRUE;
		IF NOT fbRequest.bError THEN	 
			bGetContentResult:= fbRequest.GetContent(pContent:= ADR(sContent), nContentSize:= SIZEOF(sContent), bSetNullTermination:= TRUE);
			IF fbRequest.nStatusCode >= 200 AND fbRequest.nStatusCode < 300 THEN
				bGetJsonResult:= FALSE;
				jsonDoc:= fbRequest.GetJsonDomContent(fbJson);
				IF jsonDoc <> 0 THEN
					bGetJsonResult:= TRUE;
					
					IF fbJson.HasMember(jsonDoc, 'value') THEN
					//IF fbJson.HasMember(jsonDoc, 'authenticated') THEN
					jsonVal:= fbJson.FindMember(jsonDoc, 'value');
						//jsonVal:= fbJson.FindMember(jsonDoc, 'authenticated');
						IF fbJson.IsInt(jsonVal) THEN
						//IF fbJson.IsBool(jsonVal) THEN
						//value:= fbJson.GetInt(jsonVal);
							//bResultValue:= fbJson.GetBool(jsonVal);
							nValidResCount:= nValidResCount+1;
							bError:= FALSE;						
						END_IF	
					END_IF
				END_IF							
				nResCount:= nResCount+1;			
			END_IF
		END_IF
		nState:= 0;
		bBusy:= FALSE;
		IF bError THEN
			nErrCount:= nErrCount+1;
		END_IF
	END_IF  	
END_CASE

END_FUNCTION_BLOCK

// ---- POUs/JsonSaxHandler.TcPOU
{attribute 'c++_compatible'}
FUNCTION_BLOCK JsonSaxHandler IMPLEMENTS ITcJsonSaxHandler
VAR_INPUT
END_VAR
VAR_OUTPUT
END_VAR
VAR
	(* Values from JSON - written by callback methods *)	 
	sActionID 		: STRING(80); 
	sWPID 			: STRING(80);
	iWPPlace			: DINT;
	sCell				: STRING;
	iActionType			: DINT;
	iActionState		: DINT;
	
	
	(* State machine variables *)
	eState				: E_JsonStates;
	
	(* Indicators if an expected property has been found in JSON *)
	bStartObjectFound 	: BOOL;
	bEndObjectFound		: BOOL;
	bValuesFound 		: BOOL;
	bActionIDFound 	: BOOL;
	bActionIDValueFound: BOOL;
	bWPIDFound 	: BOOL;
	bWPIDValueFound: BOOL;
	bWPPlaceFound 		: BOOL;
	bWPPlaceValueFound	: BOOL;
	bCellFound 		: BOOL;
	bCellValueFound	: BOOL;
	bActionTypeFound 		: BOOL;
	bActionTypeValueFound	: BOOL;
	bActionStateFound 		: BOOL;
	bActionStateValueFound	: BOOL;
	
	(* Error indicators *)
	bError				: BOOL;
	sErrorMsg			: STRING(255);
END_VAR

IF bError THEN
	sErrorMsg := 'JSON message does not equal expected format';
END_IF

METHOD GetActionID : STRING(80)
VAR_INPUT
END_VAR
GetActionID := sActionID;
END_METHOD

METHOD GetActionState : HRESULT
VAR_INPUT
END_VAR
GetActionState := iActionState;
END_METHOD

METHOD GetActionType : DINT
VAR_INPUT
END_VAR
GetActionType := iActionType;
END_METHOD

METHOD GetCell : STRING
VAR_INPUT
END_VAR
GetCell := sCell;
END_METHOD

METHOD GetWPID : STRING(80)
VAR_INPUT
END_VAR
GetWPID:=sWPID;
END_METHOD

METHOD GetWPPlace : DINT
VAR_INPUT
END_VAR
GetWPPlace := iWPPlace;
END_METHOD

METHOD IsFinished : BOOL
VAR_INPUT
END_VAR
IsFinished := (eState = E_JsonStates.JSON_STATE_FINISH);
END_METHOD

{attribute 'show'}
{attribute 'c++_compatible'}
{attribute 'minimal_input_size' := '4'}
{attribute 'pack_mode' := '4'}
{warning 'add method implementation'}
METHOD OnBool : HRESULT
VAR_INPUT
	value	: BOOL;
END_VAR
END_METHOD

{attribute 'show'}
{attribute 'c++_compatible'}
{attribute 'minimal_input_size' := '4'}
{attribute 'pack_mode' := '4'}
{warning 'add method implementation'}
METHOD OnDint : HRESULT
VAR_INPUT
	value	: DINT;
END_VAR

VAR

END_VAR
END_METHOD

{attribute 'show'}
{attribute 'c++_compatible'}
{attribute 'minimal_input_size' := '4'}
{attribute 'pack_mode' := '4'}
{warning 'add method implementation'}
METHOD OnEndArray : HRESULT
VAR_INPUT
	elementCount	: UDINT;
END_VAR
END_METHOD

{attribute 'show'}
{attribute 'c++_compatible'}
{attribute 'minimal_input_size' := '4'}
{attribute 'pack_mode' := '4'}
{warning 'add method implementation'}
METHOD OnEndObject : HRESULT
VAR_INPUT
	memberCount	: UDINT;
END_VAR
IF (eState = 1100) THEN
	bEndObjectFound := TRUE;
	eState := 1200;  
	ELSE

			bError := TRUE;  
END_IF
END_METHOD

{attribute 'show'}
{attribute 'c++_compatible'}
{attribute 'minimal_input_size' := '4'}
{attribute 'pack_mode' := '4'}
{warning 'add method implementation'}
METHOD OnKey : HRESULT
VAR_IN_OUT CONSTANT
	key	: STRING;
END_VAR
VAR_INPUT
	len	: UDINT;
END_VAR
IF ((eState = 11)AND(key = 'm_sActionID')) THEN
	bActionIDFound := TRUE;
	eState := 12;
ELSE
 
	IF ((eState = 20)AND(key = 'm_sWPID')) THEN
		bWPIDFound := TRUE;
		eState := 40;
	ELSE
		IF ((eState = 50)AND(key = 'm_iWPPlace')) THEN
		  bWPPlaceFound := TRUE;
		  eState := 60;
		ELSE
			IF ((eState = 70)AND(key = 'm_sCell')) THEN
				bCellFound := TRUE;
				eState := 80;
			ELSE
				IF ((eState = 90)AND(key = 'm_eActionType')) THEN
					bActionTypeFound := TRUE;
					eState := 100;
				ELSE
					IF((eState = 110)AND(key = 'm_iActionState')) THEN
					bActionStateFound := TRUE;
					eState := 120;
					ELSE

						bError := TRUE;
						Onkey := S_FALSE;
						
					END_IF

				END_IF				  
			END_IF	  
	  	END_IF
	END_IF
END_IF
END_METHOD

{attribute 'show'}
{attribute 'c++_compatible'}
{attribute 'minimal_input_size' := '4'}
{attribute 'pack_mode' := '4'}
{warning 'add method implementation'}
METHOD OnLint : HRESULT
VAR_INPUT
	value	: LINT;
END_VAR
END_METHOD

{attribute 'show'}
{attribute 'c++_compatible'}
{attribute 'minimal_input_size' := '4'}
{attribute 'pack_mode' := '4'}
{warning 'add method implementation'}
METHOD OnLreal : HRESULT
VAR_INPUT
	value	: LREAL;
END_VAR
END_METHOD

{attribute 'show'}
{attribute 'c++_compatible'}
{attribute 'minimal_input_size' := '4'}
{attribute 'pack_mode' := '4'}
{warning 'add method implementation'}
METHOD OnNull : HRESULT
END_METHOD

{attribute 'show'}
{attribute 'c++_compatible'}
{attribute 'minimal_input_size' := '4'}
{attribute 'pack_mode' := '4'}
{warning 'add method implementation'}
METHOD OnRawNumber : HRESULT
VAR_IN_OUT CONSTANT
	value	: STRING;
END_VAR
VAR_INPUT
	len	: UDINT;
END_VAR
END_METHOD

{attribute 'show'}
{attribute 'c++_compatible'}
{attribute 'minimal_input_size' := '4'}
{attribute 'pack_mode' := '4'}
{warning 'add method implementation'}
METHOD OnStartArray : HRESULT
END_METHOD

{attribute 'show'}
{attribute 'c++_compatible'}
{attribute 'minimal_input_size' := '4'}
{attribute 'pack_mode' := '4'}
{warning 'add method implementation'}
METHOD OnStartObject : HRESULT
IF (eState = 10) THEN
	bStartObjectFound := TRUE;
	eState := 11;  
ELSE

	bError := TRUE;  
			
END_IF
END_METHOD

{attribute 'show'}
{attribute 'c++_compatible'}
{attribute 'minimal_input_size' := '4'}
{attribute 'pack_mode' := '4'}
{warning 'add method implementation'}
METHOD OnString : HRESULT
VAR_IN_OUT CONSTANT
	value	: STRING;
END_VAR
VAR_INPUT
	len	: UDINT;
END_VAR

VAR
	bTimestampValueFound: BOOL;
END_VAR
IF (eState = 12)THEN
		bActionIDValueFound := TRUE;
		sActionID := value;	
		eState := 20;
ELSE
	IF (eState = 40) THEN
		bWPIDValueFound := TRUE;
		sWPID := value;
		eState := 50;
	ELSE
			IF (eState = 80) THEN
				bCellValueFound := TRUE;
				sCell :=  value ;
				eState := 90;
			ELSE
		bError := TRUE;
		OnString := S_FALSE;
		END_IF	
	END_IF
END_IF
END_METHOD

{attribute 'show'}
{attribute 'c++_compatible'}
{attribute 'minimal_input_size' := '4'}
{attribute 'pack_mode' := '4'}
{warning 'add method implementation'}
METHOD OnUdint : HRESULT
VAR_INPUT
	value	: UDINT;
END_VAR
IF (eState = 60) THEN
	bWPPlaceValueFound := TRUE;
	iWPPlace := UDINT_TO_DINT( value );
	eState := 70;
ELSE

		IF (eState = 100) THEN
			bActionTypeValueFound := TRUE;
			iActionType := UDINT_TO_DINT( value );
			eState := 110;
		ELSE
			IF (eState = 120) THEN
				bActionStateValueFound := TRUE;
				iActionState := UDINT_TO_DINT( value);
				eState := 1100;
			ELSE
				bError := TRUE;
				//OnUdint := S_FALSE;
			END_IF				
		END_IF
END_IF
END_METHOD

{attribute 'show'}
{attribute 'c++_compatible'}
{attribute 'minimal_input_size' := '4'}
{attribute 'pack_mode' := '4'}
{warning 'add method implementation'}
METHOD OnUlint : HRESULT
VAR_INPUT
	value	: ULINT;
END_VAR
END_METHOD

METHOD Reset : HRESULT
VAR_INPUT
END_VAR
	(* State machine variables *)
	eState				:= 10;
	
	(* Indicators if an expected property has been found in JSON *)
	bStartObjectFound 	:= FALSE;
	bEndObjectFound		:= FALSE;
	bValuesFound 		:= FALSE;
	bActionIDFound 		:= FALSE;
	bActionIDValueFound	:= FALSE;
	bWPIDFound 			:= FALSE;
	bWPIDValueFound		:= FALSE;
	bWPPlaceFound 		:= FALSE;
	bWPPlaceValueFound	:= FALSE;
	bCellFound 			:= FALSE;
	bCellValueFound		:= FALSE;
	bActionTypeFound 		:= FALSE;
	bActionTypeValueFound	:= FALSE;
	bActionStateFound 		:= FALSE;
	bActionStateValueFound	:= FALSE;
	
	(* Error indicators *)
	bError				:= FALSE;
END_METHOD

{attribute 'show'}
{attribute 'c++_compatible'}
{attribute 'minimal_input_size' := '4'}
{attribute 'pack_mode' := '4'}
{warning 'add method implementation'}
METHOD TcAddRef : UDINT
END_METHOD

{attribute 'show'}
{attribute 'c++_compatible'}
{attribute 'minimal_input_size' := '4'}
{attribute 'pack_mode' := '4'}
{warning 'add method implementation'}
METHOD TcQueryInterface : HRESULT
VAR_INPUT
	iid	: REFERENCE TO IID;
	pipItf	: POINTER TO PVOID;
END_VAR
END_METHOD

{attribute 'show'}
{attribute 'c++_compatible'}
{attribute 'minimal_input_size' := '4'}
{attribute 'pack_mode' := '4'}
{warning 'add method implementation'}
METHOD TcRelease : UDINT
END_METHOD

END_FUNCTION_BLOCK
